(* PLC project PlcMain, Beckhoff Automation GmbH TwinCAT PLC Control 3.5.13.21 *)
(* stored: creationDateTime 2022-08-19T12:34:24.5184426, modificationDateTime 2022-08-19T12:34:24.5184426 *)

{attribute 'qualified_only'}
{attribute 'strict'}
TYPE StateMan :
(
	Off := 0,
	Reset,
	PowerUp,
	Homing,
	Halt,
	MoveAway,
	Ready,
	Moving,
	Done
);
END_TYPE
